(* PLC project CabinetSetpointControl, Oliver Mechatronics CODESYS 3.5 *)
(* stored: creationDateTime 2026-07-14T00:00:00, modificationDateTime 2026-07-14T00:00:00 *)

(* Sequencer states for FB_CabinetSetpointControl - write -> confirm -> latch flow of a single supervisory setpoint change to the Watlow F4S over Modbus. *)
TYPE E_SetpointState : (IDLE := 0, READY := 10, WRITING := 20, CONFIRM := 30, FAULTED := 99) INT;
END_TYPE

(* Single, prioritised fault/warning code surfaced to the HMI so the operator sees a clear reason when a setpoint change is refused or the link is unhealthy. *)
TYPE E_FaultCode : (NO_FAULT := 0, COMMS_TIMEOUT := 1, WRITE_FAILED := 2, NOT_ACCEPTED := 3, RANGE_LOW := 4, RANGE_HIGH := 5, OVER_TEMP := 6) INT;
END_TYPE

(* Channel-mapped raw variables that the CODESYS Modbus Serial Master channels wire onto (I/O Mapping tab). Port /dev/ttyUSB0, 19200 8N1, slave address 1 (F4S). See codesys-modbus-integration/README.md Part 3C/4. *)
PROGRAM GVL_Modbus
  VAR_GLOBAL
    wInput1Value : WORD;  (* FC03 cyclic read, offset 100 (fallback 99), length 1 -> actual temp raw (x10) *)
    wSetpoint1Read : WORD;  (* FC03 read-back, offset 300 (fallback 299), length 1 -> SP1 raw read (x10) *)
    wSetpoint1Write : WORD;  (* FC06 write single register, offset 300 -> SP1 raw write (x10) *)
    xWriteTrigger : BOOL;  (* Rising-edge trigger var for the FC06 channel (I/O Mapping tab) *)
    xModbusError : BOOL;  (* Modbus_Slave_COM.xError *)
    xModbusDone : BOOL;  (* last transaction done *)
  END_VAR


END_PROGRAM

(* Every tag the WebVisu screen binds to. Gear button opens a pop-up (dlgSetpoint) bound to rReqSetpoint / xSetBtn / xResetBtn. See codesys-modbus-integration/README.md. *)
PROGRAM GVL_HMI
  VAR_GLOBAL
    rChamberTemp : REAL;  (* actual temp, deg C (read/10) *)
    rConfirmedSetpoint : REAL;  (* last confirmed SP, deg C *)
    rReqSetpoint : REAL := 75.0;  (* operator entry (dialog), deg C *)
    xSetBtn : BOOL;  (* dialog SET button *)
    xResetBtn : BOOL;  (* dialog/banner RESET button *)
    xSetpointConfirmed : BOOL;  (* green banner driver *)
    xFaultActive : BOOL;  (* red banner driver *)
    eFaultCode : E_FaultCode;
    sStatusText : STRING(80);
  END_VAR


END_PROGRAM

(* Supervisory setpoint control for the Left Hand Small Temperature Cabinet (Watlow F4S, Modbus RTU / RS-232). Reads/writes GVL_Modbus and GVL_HMI directly in its body per the Project Development Package spec - see the .st source header for the known follow-up note on this coupling. *)
FUNCTION_BLOCK FB_CabinetSetpointControl
  VAR
    rtrigSet : R_TRIG;  (* Edge detect on SET command *)
    rtrigReset : R_TRIG;  (* Edge detect on RESET command *)
    tonWatchdog : TON;  (* Comms-loss debounce *)
    tonConfirmWait : TON;  (* Read-back confirm timeout *)
    wTargetRaw : WORD;  (* Setpoint being written, raw x10 *)
    rReadBack : REAL;  (* Setpoint echo, engineering units *)
  END_VAR
  VAR_INPUT
    rRequestedSetpoint : REAL;  (* deg C from HMI *)
    xSetCommand : BOOL;  (* HMI SET - rising edge applies *)
    xReset : BOOL;  (* fault reset - rising edge clears *)
    xOverTempDI : BOOL;  (* spare EL1409 DI, TRUE = over-temp *)
    rMinSetpoint : REAL := 30.0;  (* Lower safe bound, degC *)
    rMaxSetpoint : REAL := 130.0;  (* Upper safe bound, degC *)
    rScale : REAL := 10.0;  (* eng <-> raw multiplier *)
    rTolerance : REAL := 0.1;  (* deg C read-back tolerance *)
    tCommsTimeout : TIME := T#3s;  (* watchdog *)
  END_VAR
  VAR_OUTPUT
    eState : E_SetpointState;
    eFault : E_FaultCode;
    xConfirmed : BOOL;
    xFault : BOOL;
    rActualTemp : REAL;  (* Live chamber temperature, degC *)
    rConfirmedSetpoint : REAL;  (* Last accepted setpoint, degC *)
  END_VAR

(* ---- Edge detect ---- *)
rtrigSet(CLK := xSetCommand);
rtrigReset(CLK := xReset);

(* ---- Always-live scaling of the cyclic read ---- *)
rActualTemp          := WORD_TO_REAL(GVL_Modbus.wInput1Value) / rScale;
rReadBack             := WORD_TO_REAL(GVL_Modbus.wSetpoint1Read) / rScale;
GVL_HMI.rChamberTemp := rActualTemp;

(* ---- Comms watchdog: LEVEL signal, NOT an edge pulse (avoids R_TRIG->TON trap) ---- *)
tonWatchdog(IN := NOT GVL_Modbus.xModbusDone, PT := tCommsTimeout);

(* ---- Over-temp interlock (highest priority latch) ---- *)
IF xOverTempDI THEN
    eFault := E_FaultCode.OVER_TEMP;
    eState := E_SetpointState.FAULTED;
END_IF

(* ---- Comms loss latch (any state) ---- *)
IF tonWatchdog.Q OR GVL_Modbus.xModbusError THEN
    eFault := E_FaultCode.COMMS_TIMEOUT;
    eState := E_SetpointState.FAULTED;
END_IF

CASE eState OF

    E_SetpointState.IDLE:
        xConfirmed := TRUE;
        GVL_Modbus.xWriteTrigger := FALSE;
        IF rtrigSet.Q THEN
            eState := E_SetpointState.READY;
        END_IF

    E_SetpointState.READY:
        xConfirmed := FALSE;
        IF rRequestedSetpoint < rMinSetpoint THEN
            eFault := E_FaultCode.RANGE_LOW;
            eState := E_SetpointState.FAULTED;
        ELSIF rRequestedSetpoint > rMaxSetpoint THEN
            eFault := E_FaultCode.RANGE_HIGH;
            eState := E_SetpointState.FAULTED;
        ELSE
            wTargetRaw := REAL_TO_WORD(rRequestedSetpoint * rScale);
            GVL_Modbus.wSetpoint1Write := wTargetRaw;
            eState := E_SetpointState.WRITING;
        END_IF

    E_SetpointState.WRITING:
        GVL_Modbus.xWriteTrigger := TRUE;    (* one-shot rising edge fires FC06 *)
        eState := E_SetpointState.CONFIRM;

    E_SetpointState.CONFIRM:
        GVL_Modbus.xWriteTrigger := FALSE;   (* drop trigger to re-arm the edge *)
        tonConfirmWait(IN := TRUE, PT := tCommsTimeout);
        IF ABS(rReadBack - rRequestedSetpoint) <= rTolerance THEN
            rConfirmedSetpoint := rReadBack;
            GVL_HMI.rConfirmedSetpoint := rReadBack;
            tonConfirmWait(IN := FALSE);
            eState := E_SetpointState.IDLE;
        ELSIF tonConfirmWait.Q THEN
            eFault := E_FaultCode.NOT_ACCEPTED;
            eState := E_SetpointState.FAULTED;
        END_IF

    E_SetpointState.FAULTED:
        xConfirmed := FALSE;
        GVL_Modbus.xWriteTrigger := FALSE;
        (* Latched - clears only on reset edge AND only if condition is gone *)
        IF rtrigReset.Q
           AND NOT xOverTempDI
           AND NOT tonWatchdog.Q
           AND NOT GVL_Modbus.xModbusError THEN
            eFault := E_FaultCode.NO_FAULT;
            eState := E_SetpointState.IDLE;
        END_IF

END_CASE

xFault                      := (eState = E_SetpointState.FAULTED);
GVL_HMI.xSetpointConfirmed  := xConfirmed AND NOT xFault;
GVL_HMI.xFaultActive        := xFault;
GVL_HMI.eFaultCode          := eFault;
END_FUNCTION_BLOCK

(* Cyclic entry point (MainTask). xOverTempDI is wired to GVL_Modbus.xModbusError as a placeholder - REPLACE with the real mapped EL1409 digital-input channel before relying on this interlock. *)
PROGRAM PLC_PRG
  VAR
    fbSetpoint : FB_CabinetSetpointControl;
  END_VAR

(* ---- Drive the supervisory setpoint controller ---- *)
fbSetpoint(
    rRequestedSetpoint := GVL_HMI.rReqSetpoint,
    xSetCommand        := GVL_HMI.xSetBtn,
    xReset             := GVL_HMI.xResetBtn,
    xOverTempDI        := GVL_Modbus.xModbusError,  (* REPLACE with mapped EL1409 DI channel *)
    rMinSetpoint       := 30.0,
    rMaxSetpoint       := 130.0
);

(* ---- Consume dialog button one-shots ---- *)
GVL_HMI.xSetBtn   := FALSE;
GVL_HMI.xResetBtn := FALSE;
END_PROGRAM
